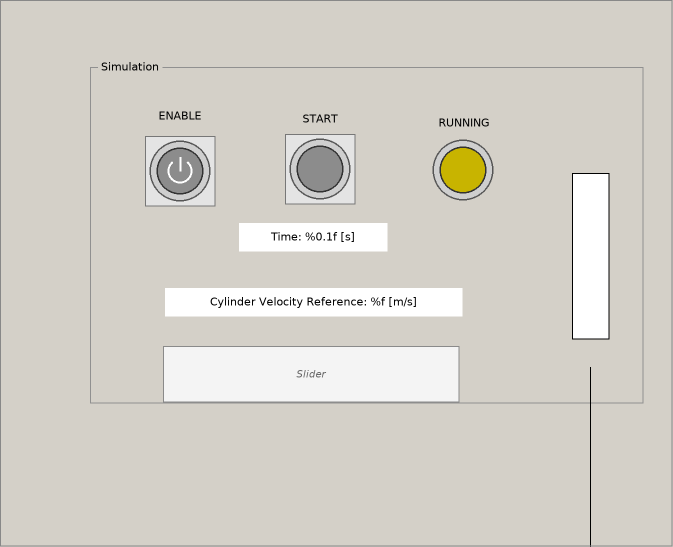
VISUALIZATION CraneHMI  // 673x547
    Rectangle (507,238 166x37), angle 270
        p2738717112: Outputs.fCylinderPosition
    GroupBox (90,59 553x344), "Simulation"
        PowerSwitch (55,77 70x70), variable: Inputs.bEnableSimulation, behaviour: TOGGLE, style: Switch-PowerSwitch-Gray
        PushSwitch (195,75 70x70), variable: Inputs.bStartSimulation, behaviour: TOGGLE, style: Switch-PushSwitch-Gray
        Lamp1 (338,76 70x70), variable: Outputs.bSimulationRunning, style: Lamp-Lamp1-Yellow
        Textfield (74,228 299x30), "Cylinder Velocity Reference: %f [m/s]", text variable: Inputs.fCylinderVelocityReference
            OnMouseClick: write the text variable via Default
        Label (15,42 150x30), "ENABLE"
        Label (155,45 150x30), "START"
        Label (299,49 150x30), "RUNNING"
        Textfield (148,163 150x30), "Time: %0.1f [s]", text variable: Outputs.fSimulationTime
        Slider (73,287 296x56), variable: Inputs.fCylinderVelocityReference, scale -0.1..0.1
    Line (590,367) (590,547)
        p1126004900: Outputs.pt1_y
        p3528305787: Outputs.pt0_x
        p2773130477: Outputs.pt0_y
        p874137650: Outputs.pt1_x
END_VISUALIZATION

(* stored: Version 1.1.0.1, ProductVersion 3.1.4024.9
   Visu CraneHMI: Id {4bdd8ed7-7379-4dd1-955f-a8a1c50d5ff4} *)
